//散配區座標結構
TYPE st_AllocateParameterCore  :
STRUCT
  	fName  :STRING;
 	index:  LREAL;
	X      :LREAL;
	Y      :LREAL;
	Clip   :LREAL;
	Excute:BOOL;
	Done  :BOOL;
END_STRUCT
END_TYPE

(* stored: Version 1.1.0.1, ProductVersion 3.1.4024.13
   DUT st_AllocateParameterCore: Id {e650a918-2ce7-4bf9-b364-1718667cc3bb} *)
